Staubli VAL3: NUM.dtx

public string sItems
num nIndex
string sMessage
num nMode
